{attribute 'GeneratedUsingTerminal: EL5151-0021-0018'}
{attribute addProperty BoxType "EL5151-0021-0018"}
{attribute addProperty Id "Latch_C_validBOOL1Latch_extern_validBOOL1Set_counter_doneBOOL1Measurement_doneBOOL1Status_of_input_ABOOL1Status_of_input_BBOOL1Status_of_input_CBOOL1Status_of_outputBOOL1Status_of_extern_latchBOOL1Compatible_input_cycle_counter_highBOOL1TxPDO_ToggleBOOL1"}
{attribute addProperty CRC "1004781350"}
{attribute addProperty Size "11"}
TYPE Status_3BE3BF26 :
STRUCT
	{attribute addProperty Name "Latch_C_valid"}
	Latch_C_valid : BOOL;
	{attribute addProperty Name "Latch_extern_valid"}
	Latch_extern_valid : BOOL;
	{attribute addProperty Name "Set_counter_done"}
	Set_counter_done : BOOL;
	{attribute addProperty Name "Measurement_done"}
	Measurement_done : BOOL;
	{attribute addProperty Name "Status_of_input_A"}
	Status_of_input_A : BOOL;
	{attribute addProperty Name "Status_of_input_B"}
	Status_of_input_B : BOOL;
	{attribute addProperty Name "Status_of_input_C"}
	Status_of_input_C : BOOL;
	{attribute addProperty Name "Status_of_output"}
	Status_of_output : BOOL;
	{attribute addProperty Name "Status_of_extern_latch"}
	Status_of_extern_latch : BOOL;
	{attribute addProperty Name "Compatible_input_cycle_counter_high"}
	Compatible_input_cycle_counter_high : BOOL;
	{attribute addProperty Name "TxPDO_Toggle"}
	TxPDO_Toggle : BOOL;
END_STRUCT
END_TYPE

(* stored: Version 1.2.0.0, ProductVersion 3.1.4024.9
   DUT Status_3BE3BF26: Id {f3e76544-474f-4230-b221-860627fe012a} *)
